// TwinCAT 3 PLC project Untitled1
// ProgramVersion: 3.1.4024.0
// libraries:
//   Tc2_Standard, * (Beckhoff Automation GmbH)
//   Tc2_System, * (Beckhoff Automation GmbH)
//   Tc3_Module, * (Beckhoff Automation GmbH)
// project tree:
//   / PlcTask.TcTTO
//   POUs/ MAIN.TcPOU
// real-time tasks:
//   TASK PlcTask: cycle T#10ms, priority 20, ADS port 350

CONFIGURATION Untitled1
    RESOURCE PLC ON TwinCAT3
        TASK PlcTask(INTERVAL := T#10ms, PRIORITY := 20);
        PROGRAM MAIN WITH PlcTask : MAIN;
    END_RESOURCE
END_CONFIGURATION

// ---- POUs/MAIN.TcPOU
PROGRAM MAIN
VAR
	Timer : TON;
	
	Start : BOOL;
	inTime : TIME := T#1h10m10s;
	
	Done : BOOL;
	outTime : TIME;
	
	RemainingTime : TIME;
	Reset : BOOL;
END_VAR

Timer(IN:=Start, PT:=inTime, Q=>Done, ET=>outTime);
RemainingTime := inTime - outTime;

IF Reset THEN
	Start := FALSE;
	Reset := FALSE;
END_IF

END_PROGRAM
